{attribute 'linkalways'} 
{attribute 'no_explicit_call' := 'This FB is a CLASS and must be accessed using methods or properties'}
{attribute 'enable_dynamic_creation'}
FUNCTION_BLOCK SequentialResponseIdGenerator IMPLEMENTS I_ResponseIdGenerator
VAR
	currentCount : UDINT;
END_VAR

METHOD PUBLIC Generate : T_MAXSTRING
VAR_INPUT
END_VAR
currentCount := currentCount + 1;
Generate := UDINT_TO_STRING(currentCount);
END_METHOD

END_FUNCTION_BLOCK

(* stored: Version 1.1.0.1, ProductVersion 3.1.4024.12
   POU SequentialResponseIdGenerator: Id {011a3733-d36c-05de-113c-bb069ea776cf}, SpecialFunc None
   Method Generate: Id {9d94b21d-b6a5-0e68-0f20-647f267a9048} *)
